// TIA Portal V17 export
// export: Created 2025-03-05T07:59:02.0903063Z, ExportSetting WithDefaults, DisplayName Totally Integrated Automation Portal, DisplayVersion V17 Update 8, DisplayName TIA Portal Openness, DisplayVersion V17 Update 8, DisplayName TIA Portal Version Control Interface, DisplayVersion V17, DisplayName SINAMICS Startdrive Advanced, DisplayVersion V17 SP2, DisplayName SINAMICS Startdrive G110M, G120, G120C, G120D, G120P, G115D, DisplayVersion V17 SP2, DisplayName SINAMICS Startdrive G130, G150, S120, S150, SINAMICS MV, S210, DisplayVersion V17 SP2, DisplayName STEP 7 Professional, DisplayVersion V17 Update 8, DisplayName SINUMERIK ONE STEP 7 Toolbox, DisplayVersion V17 Update 12, DisplayName SINUMERIK 840D sl STEP 7 Toolbox, DisplayVersion V17 Update 12, DisplayName STEP 7 Safety, DisplayVersion V17 Update 6, DisplayName WinCC Advanced, DisplayVersion V17 Update 8
DATA_BLOCK "DB2430_FULL_DEPTH"   // DB2430
{ S7_Optimized_Access := 'FALSE'; DB_Accessible_From_OPC_UA := 'FALSE' }
AUTHOR : ETXETAR
VERSION : 1.0
// stored: AutoNumber false, DBAccessibleFromOPCUA false, DBAccessibleFromWebserver true, IsOnlyStoredInLoadMemory false, IsWriteProtectedInAS false
   VAR RETAIN
      FD_UNIT_01 : Struct
         FIXTURE_1 : "FULL_DEPTH_CLADDING";
         FIXTURE_2 : "FULL_DEPTH_CLADDING";
         FIXTURE_3 : "FULL_DEPTH_CLADDING";
         FIXTURE_4 : "FULL_DEPTH_CLADDING";
         FIX_IN_STA_1_FD { S7_SetPoint := 'True'} : Bool;   // FIXTURE IN UNIT 01 STATION 1 FULL DEPTH
         FIX_IN_STA_2_FD { S7_SetPoint := 'True'} : Bool;   // FIXTURE IN UNIT 01 STATION 2 FULL DEPTH
         FIX_IN_STA_3_FD { S7_SetPoint := 'True'} : Bool;   // FIXTURE IN UNIT 01 STATION 3 FULL DEPTH
         FIX_IN_STA_4_FD { S7_SetPoint := 'True'} : Bool;   // FIXTURE IN UNIT 01 STATION 4 FULL DEPTH
      END_STRUCT;
      FD_UNIT_02 : Struct
         FIXTURE_1 : "FULL_DEPTH_CLADDING";
         FIXTURE_2 : "FULL_DEPTH_CLADDING";
         FIXTURE_3 : "FULL_DEPTH_CLADDING";
         FIXTURE_4 : "FULL_DEPTH_CLADDING";
         FIX_IN_STA_1_FD { S7_SetPoint := 'True'} : Bool;   // FIXTURE IN UNIT 02 STATION 1 FULL DEPTH
         FIX_IN_STA_2_FD { S7_SetPoint := 'True'} : Bool;   // FIXTURE IN UNIT 02 STATION 2 FULL DEPTH
         FIX_IN_STA_3_FD { S7_SetPoint := 'True'} : Bool;   // FIXTURE IN UNIT 02 STATION 3 FULL DEPTH
         FIX_IN_STA_4_FD { S7_SetPoint := 'True'} : Bool;   // FIXTURE IN UNIT 02 STATION 4 FULL DEPTH
      END_STRUCT;
      FD_UNIT_03 : Struct
         FIXTURE_1 : "FULL_DEPTH_CLADDING";
      END_STRUCT;
   END_VAR
BEGIN
END_DATA_BLOCK
